(*
Nazwa:			FB_State
Opis:			Generowanie stanów 
Wersja:			v1.0
Data:			2020-04-14
Autor:			DP
Urzadzenia:		
Konfiguracja:	
Info: 
*)

FUNCTION_BLOCK FB_State
VAR_INPUT
	eState							:E_Station;						//Stan ogólny bloku
	bRun							:BOOL;							//Rozkad cyklu	
	eGripperScrewerRunningState		:E_GripperScrewer; 				//Stan zakręcarki szczekowej							
	//eRollerScrewerRunningState		:E_RollerScrewer; 				//Stan zakręcarki rolkowej						
	eCheckerRunningState			:E_CheckerState; 				//Stan sprawdzania
	eEntranceGatesRunningState		:E_EntranceGatesState;			//Stan szlabanów
	eCatchRunningState				:E_CatchStationState;			//Stan wewnętrzny
	eCapPushingRunningState			:E_CapPushingState;				//Stan wbijaka
	eMassHeatingRunningState		:E_MassHeatingState;			//Stan grzania
	eConveyorRunningState			:E_ConveyorState;				//Stan transprterów
	eFormsDragingRunningState 		:E_DragStationState;				//Stan przeciągania zwykłego
	eFormsDragingPneumRunningState	:E_DragStationStatePneum;
	eLidSealingRunningState			:E_LidSealing;					//Stan zgrzewania
	eLidFeederRunningState			:E_LidFeederState;				//Stan platynkowania
	//eWheelRunningState				:E_WheelState;					//Stan kola
	eDispencerRunningState			:E_DispencerState;				//Stan dozowników
	eDispencerLifterRunningState	:E_DispencerLifterState;		//Stan podnośnikow
	eCapFeederRobotRunningState		:E_RobotMovState;				//Stan robota
	eWeightRunningState				:E_WeightState;	
	eWeightLiftRunningState			:E_WeightLiftStationState	;	//Stan wagi		
	eBottleSorterRunningState		:E_BottleFeederState;			// Stan podajnik opakowań		 
	eCapFeederRunningState			:E_CapFeederState;				//Stan podajnika nasadek			
	eWickFeederRunningState			:E_WickFeederState;
END_VAR
VAR_OUTPUT
	sStateDesc						:STRING;
	iState							:INT;							//Stan ogólny bloku
END_VAR
VAR
	iC: INT;
	i: E_DispencerState;
	ic2: INT;
	ic3: INT;
	ic4: INT;
END_VAR


IF 	eState = 0 THEN // eDisabled := 0,	
	sStateDesc := 'Wyłączona';
ELSIF 	eState = 1 THEN // eAborted := 1,
	sStateDesc := 'Bezpieczne zatrzymanie';
ELSIF 	eState = 2 THEN // eAborting := 2,  
	sStateDesc := 'Bezpieczne zatrzymywanie';
ELSIF 	eState = 3 THEN // eError := 3,	
	sStateDesc := 'Błąd';
ELSIF 	eState = 4 THEN // eResetting := 4,	
	sStateDesc := 'Resetowanie';
ELSIF 	eState = 5 THEN // eManualMovement := 5, 
	sStateDesc := 'Tryb serwisowy';
ELSIF 	eState = 6 THEN // eHoming := 6,
	sStateDesc := 'Bazowanie';
ELSIF 	eState = 7 THEN // eHomingDone := 7,
	sStateDesc := 'Koniec bazowania';	
ELSIF 	eState = 8 THEN // ePreparingToReady := 8,	
	sStateDesc := 'Przygotowanie do gotowości';
ELSIF 	eState = 9 THEN // ePreparingToDisable := 9,
	sStateDesc := 'Przygotowanie do wyłączenia';	
ELSIF 	eState = 10 THEN // eReady	:= 10,
	sStateDesc := 'Gotowa';	
ELSIF 	eState = 11 THEN // eStopping := 11,
	sStateDesc := 'Zatrzymywanie';	
ELSIF 	eState = 12 THEN // eStarting := 12,
	sStateDesc := 'Uruchamianie';  
ELSIF 	eState = 13 THEN // eRunning := 13		
	sStateDesc := 'Praca';
END_IF

IF eState = 13 OR bRun THEN
	GripperScrewer();
	BottleSorter();
	RollerScrewer();	
	EntranceGates();
	CatchStation();
	MassHeating();
	Conveyor();
	CapFeeder();
	Checker();
	Dispencer();
	DispencerLifter();
	Robot();
	Weight();
	WeightLift();
	Drag();
	DragPneum();
	LidFeeder();
	LidSealing();
	WickFeeder();
END_IF

iState := eState;

ACTION BottleSorter:

IF eBottleSorterRunningState  = 1 THEN 
	sStateDesc := 'Błąd';	
ELSIF eBottleSorterRunningState  = 2 THEN 
	sStateDesc := 'Gotowa';	
ELSIF eBottleSorterRunningState  = 3 THEN 
	sStateDesc := 'Bazowanie';	
ELSIF eBottleSorterRunningState  = 4 THEN 
	sStateDesc := 'Koniec bazowania';	
ELSIF eBottleSorterRunningState  = 5 THEN 
	sStateDesc := 'Tryb ręczny';
ELSIF eBottleSorterRunningState  = 60 THEN 
	sStateDesc := 'Przygotowanie do ruchu';	
ELSIF eBottleSorterRunningState  = 70 THEN 
	sStateDesc := 'Zamknięcie bramki lewej';	
ELSIF eBottleSorterRunningState  = 80 THEN 
	sStateDesc := 'Przejazd do pobrania';	
ELSIF eBottleSorterRunningState  = 90 THEN 
	sStateDesc := 'Zamykanie chwytaka';	
ELSIF eBottleSorterRunningState  = 100 THEN 
	sStateDesc := 'Otwarcie bramki prawej';	
ELSIF eBottleSorterRunningState  = 110 THEN 
	sStateDesc := 'Przejazd nad formatke';	
ELSIF eBottleSorterRunningState  = 120 THEN 
	sStateDesc := 'Zamknięcie bramki lewej';	
ELSIF eBottleSorterRunningState  = 130 THEN 
	sStateDesc := 'Zamknięcie docisku';	
ELSIF eBottleSorterRunningState  = 140 THEN 
	sStateDesc := 'Wkładanie opakowania';	
ELSIF eBottleSorterRunningState  = 150 THEN 
	sStateDesc := 'Otwieranie chwytaka';
ELSIF eBottleSorterRunningState  = 160 THEN 
	sStateDesc := 'Powrót do pozycji gotowości';
ELSIF eBottleSorterRunningState  = 170 THEN 
	sStateDesc := 'Wypuszczanie formatki';
		
END_IF
END_ACTION

ACTION CapFeeder:
IF eCapFeederRunningState = 1 THEN
	sStateDesc := 'Gotowy';
ELSIF eCapFeederRunningState = 2 THEN
	sStateDesc := 'Niski poziom zamknięć';
ELSIF eCapFeederRunningState = 3 THEN
	sStateDesc := 'Praca';
ELSIF eCapFeederRunningState = 4 THEN
	sStateDesc := 'Zapełniony';
END_IF
END_ACTION

ACTION CapPushing:
IF eCapPushingRunningState = 1 THEN
	sStateDesc := 'Gotowy';
ELSIF eCapPushingRunningState = 2 THEN
	sStateDesc := 'Wbijanie';
ELSIF eCapPushingRunningState = 3 THEN
	sStateDesc := 'Przyciskanie';	
ELSIF eCapPushingRunningState = 4 THEN
	sStateDesc := 'Wbito';		
ELSIF eCapPushingRunningState = 5 THEN
	sStateDesc := 'Podnoszenie';									
END_IF
END_ACTION

ACTION CatchStation:
IF eCatchRunningState = 1 THEN
	sStateDesc := 'Błąd';
ELSIF eCatchRunningState = 2 THEN
	sStateDesc := 'Tryb serwisowy';
ELSIF eCatchRunningState = 4 THEN
	sStateDesc := 'Bazowanie';	
ELSIF eCatchRunningState = 5 THEN
	sStateDesc := 'Koniec bazownia';		
ELSIF eCatchRunningState = 6 THEN
	sStateDesc := 'Gotowość';			
ELSIF eCatchRunningState = 7 THEN
	sStateDesc := 'Chwytanie';				
ELSIF eCatchRunningState = 8 THEN
	sStateDesc := 'Chwycono';					
ELSIF eCatchRunningState = 9 THEN
	sStateDesc := 'Przygotowanie do wyłączenia';	
ELSIF eCatchRunningState = 10 THEN
	sStateDesc := 'Nie chwycono';					
END_IF
END_ACTION

ACTION Checker:
IF eCheckerRunningState = 1 THEN
	sStateDesc := 'Blad';
ELSIF eCheckerRunningState = 2 THEN
	sStateDesc := 'Tryb serwisowy';	
ELSIF eCheckerRunningState = 3 THEN
	sStateDesc := 'Bazowanie';		
ELSIF eCheckerRunningState = 4 THEN
	sStateDesc := 'Koniec bazowania';			
ELSIF eCheckerRunningState = 5 THEN
	sStateDesc := 'Gotowa';				
ELSIF eCheckerRunningState = 6 THEN
	sStateDesc := 'Formatka';		
ELSIF eCheckerRunningState = 7 THEN
	sStateDesc := 'Butelka';	
ELSIF eCheckerRunningState = 8 THEN
	sStateDesc := 'Platynka OK';	
ELSIF eCheckerRunningState = 9 THEN
	sStateDesc := 'Nasadka OK';	
ELSIF eCheckerRunningState = 10 THEN
	sStateDesc := 'Nasadka NOK.';		
ELSIF eCheckerRunningState = 11 THEN
	sStateDesc := 'Przyg. do wył.';		
					
END_IF
END_ACTION

ACTION Conveyor:
(*IF eConveyorRunningState = 0 THEN //Wyłączona
	sStateDesc := 'Wyłączona';
ELSIF eConveyorRunningState = 1 THEN //Błąd
	sStateDesc := 'Bład';
ELSIF eConveyorRunningState = 2 THEN //Tryb serwisowy
	sStateDesc := 'Tryb serwisowy';	
ELSIF eConveyorRunningState = 3 THEN //Bazowanie
	sStateDesc := 'Bazowanie';		
ELSIF eConveyorRunningState = 4 THEN //Koniec bazowania
	sStateDesc := 'Koniec bazowanie';	
ELSIF eConveyorRunningState = 5 THEN //gotowość
	sStateDesc := 'Gotowa';	
ELSIF eConveyorRunningState = 6 THEN //Zatrzymywanie
	sStateDesc := 'Zatrzymywanie';	
ELSIF eConveyorRunningState = 7 THEN //Startowanie
	sStateDesc := 'Startowanie';	
ELSIF eConveyorRunningState = 8 THEN //Praca
	sStateDesc := 'Praca';				
END_IF


*)
(*
IF eConveyorRunningState = 0 THEN //Wyłączona
	sStateDesc := 'Wyłączona 123';
ELSIF eConveyorRunningState = 1 THEN //Błąd
	sStateDesc := 'Bezp. zatrzymana';
ELSIF eConveyorRunningState = 2 THEN //Tryb serwisowy
	sStateDesc := 'Bezp. zatrzymywanie';	
ELSIF eConveyorRunningState = 3 THEN //Bazowanie
	sStateDesc := 'Błąd';		
ELSIF eConveyorRunningState = 4 THEN //Koniec bazowania
	sStateDesc := 'Resetowanie błędów';	
ELSIF eConveyorRunningState = 5 THEN //gotowość
	sStateDesc := 'Tryb ręczny';	
ELSIF eConveyorRunningState = 6 THEN //Zatrzymywanie
	sStateDesc := 'Bazowanie';	
ELSIF eConveyorRunningState = 7 THEN //Startowanie
	sStateDesc := 'Koniec bazowania';	
ELSIF eConveyorRunningState = 8 THEN //Praca
	sStateDesc := 'Przyg. do wył.';	
	*)
IF eConveyorRunningState = 10 THEN //Startowanie
	sStateDesc := 'Gotowośc';	
ELSIF eConveyorRunningState = 11 THEN //Praca
	sStateDesc := 'Zatrzymywanie';	
ELSIF eConveyorRunningState = 12 THEN //Praca
	sStateDesc := 'Uruchamianie';	
ELSIF eConveyorRunningState = 13 THEN //Praca
	sStateDesc := 'Praca';

	
END_IF
END_ACTION

ACTION Dispencer:
IF eDispencerRunningState = 5 THEN
	sStateDesc := 'Gotowa';	
		ic3		:= ic3+1;		
ELSIF eDispencerRunningState = 6 THEN
	sStateDesc := 'Przyg. dozy';		
ELSIF eDispencerRunningState = 7 THEN
	sStateDesc := '1 faza';	
ELSIF eDispencerRunningState = 8 THEN
	sStateDesc := '2 faza';	
ELSIF eDispencerRunningState = 9 THEN
	sStateDesc := '3 faza';	
ELSIF eDispencerRunningState = 10 THEN
	sStateDesc := 'Koniec dozy';	
ELSIF eDispencerRunningState = 11 THEN
	sStateDesc := 'Podsys';	
ELSIF eDispencerRunningState = 12 THEN
	sStateDesc := 'Koniec pods.';	
ELSIF eDispencerRunningState = 13 THEN
	sStateDesc := 'Zasysanie';				
ELSIF eDispencerRunningState = 14 THEN
	sStateDesc := 'Podnoszenie';	
ELSIF eDispencerRunningState = 15 THEN
	sStateDesc := 'Przerywanie';			
ELSIF eDispencerRunningState = 16 THEN
	sStateDesc := 'Przyg. do wył.';	
ELSIF eDispencerRunningState = 17 THEN
	sStateDesc := 'Przeciąganie';
ELSIF eDispencerRunningState = 18 THEN
	sStateDesc := 'Przyg. do mycia';
ELSIF eDispencerRunningState = 19 THEN
	sStateDesc := 'Gotowy do mycia';
ELSIF eDispencerRunningState = 20 THEN
	sStateDesc := 'Mycie';
ELSIF eDispencerRunningState = 21 THEN
	sStateDesc := 'Koniec mycia';		
END_IF

i   := eDispencerRunningState;
END_ACTION

ACTION DispencerLifter:
IF eDispencerLifterRunningState = 1 THEN
	sStateDesc := 'Blad';
ELSIF eDispencerLifterRunningState = 2 THEN
	sStateDesc := 'Tryb serwisowy';	
ELSIF eDispencerLifterRunningState = 3 THEN
	sStateDesc := 'Bazowanie';		
ELSIF eDispencerLifterRunningState = 4 THEN
	sStateDesc := 'Koniec bazowania';			
ELSIF eDispencerLifterRunningState = 5 THEN
	sStateDesc := 'Gotowa';				
ELSIF eDispencerLifterRunningState = 6 THEN
	sStateDesc := 'Przyg. dozy';		
ELSIF eDispencerLifterRunningState = 7 THEN
	sStateDesc := '1 faza';	
ELSIF eDispencerLifterRunningState = 8 THEN
	sStateDesc := '2 faza';	
ELSIF eDispencerLifterRunningState = 9 THEN
	sStateDesc := '3 faza';	
ELSIF eDispencerLifterRunningState = 10 THEN
	sStateDesc := 'Koniec dozy';	
ELSIF eDispencerLifterRunningState = 11 THEN
	sStateDesc := 'Zasysanie';	
ELSIF eDispencerLifterRunningState = 12 THEN
	sStateDesc := 'Podnoszenie';	
ELSIF eDispencerLifterRunningState = 13 THEN
	sStateDesc := 'Wylaczanie';				
ELSIF eDispencerLifterRunningState = 14 THEN
	sStateDesc := 'Przyg. do wył.';	
ELSIF eDispencerLifterRunningState = 15 THEN
	sStateDesc := 'Przeciąganie';			
ELSIF eDispencerLifterRunningState = 16 THEN
	sStateDesc := 'Podsysanie';	
ELSIF eDispencerLifterRunningState = 17 THEN
	sStateDesc := 'Koniec podsysania';		
END_IF
END_ACTION

ACTION Drag:
IF eFormsDragingRunningState = 1 THEN 
	sStateDesc := 'Bład';
ELSIF eFormsDragingRunningState  = 2 THEN 
	sStateDesc := 'Gotowość';	
ELSIF eFormsDragingRunningState  = 3 THEN 
	sStateDesc := 'Tryb serwisowy';	
ELSIF eFormsDragingRunningState  = 4 THEN 
	sStateDesc := 'Przygotowanie do ruchu';	
ELSIF eFormsDragingRunningState  = 5 THEN 
	sStateDesc := 'Bazowanie';	
ELSIF eFormsDragingRunningState  = 6 THEN 
	sStateDesc := 'Koniec bazowania';	
ELSIF eFormsDragingRunningState  = 7 THEN 
	sStateDesc := 'Podnoszenie';	
ELSIF eFormsDragingRunningState  = 8 THEN 
	sStateDesc := 'Przyg. do przec.';	
ELSIF eFormsDragingRunningState  = 9 THEN 
	sStateDesc := 'Przeciąganie';	
ELSIF eFormsDragingRunningState  = 10 THEN 
	sStateDesc := 'Koniec Przec.';	
ELSIF eFormsDragingRunningState  = 11 THEN 
	sStateDesc := 'Zakańczanie przec.';	
ELSIF eFormsDragingRunningState  = 12 THEN 
	sStateDesc := 'Koniec zakań. przec.';	
ELSIF eFormsDragingRunningState  = 13 THEN 
	sStateDesc := 'Opuszczanie';	
ELSIF eFormsDragingRunningState  = 14 THEN 
	sStateDesc := 'Przeciągniete';	
ELSIF eFormsDragingRunningState  = 15 THEN 
	sStateDesc := 'Koniec cyklu';	
			
END_IF
END_ACTION

ACTION DragPneum:
IF eFormsDragingPneumRunningState= 1 THEN 
	sStateDesc := 'Bład';
ELSIF eFormsDragingPneumRunningState  = 2 THEN 
	sStateDesc := 'Gotowość';	
ELSIF eFormsDragingPneumRunningState  = 3 THEN 
	sStateDesc := 'Tryb serwisowy';	
ELSIF eFormsDragingPneumRunningState  = 4 THEN 
	sStateDesc := 'Przygotowanie do ruchu';	
ELSIF eFormsDragingPneumRunningState  = 5 THEN 
	sStateDesc := 'Bazowanie';	
ELSIF eFormsDragingPneumRunningState  = 6 THEN 
	sStateDesc := 'Koniec bazowania';	
ELSIF eFormsDragingPneumRunningState  = 7 THEN 
	sStateDesc := 'Podnoszenie';	
ELSIF eFormsDragingPneumRunningState  = 8 THEN 
	sStateDesc := 'Przyg. do przec.';	
ELSIF eFormsDragingPneumRunningState  = 9 THEN 
	sStateDesc := 'Przeciąganie';	
ELSIF eFormsDragingPneumRunningState  = 10 THEN 
	sStateDesc := 'Koniec Przec.';	
ELSIF eFormsDragingPneumRunningState  = 11 THEN 
	sStateDesc := 'Korekta pozycji';	
ELSIF eFormsDragingPneumRunningState  = 12 THEN 
	sStateDesc := 'Koniec korekty';	
ELSIF eFormsDragingPneumRunningState  = 13 THEN 
	sStateDesc := 'Opuszczanie';	
ELSIF eFormsDragingPneumRunningState  = 14 THEN 
	sStateDesc := 'Przeciągniete';	
ELSIF eFormsDragingPneumRunningState  = 15 THEN 
	sStateDesc := 'Koniec cyklu';					
END_IF
END_ACTION

ACTION EntranceGates:
IF eEntranceGatesRunningState = 1 THEN
	sStateDesc := 'Błąd';
ELSIF eEntranceGatesRunningState = 2 THEN
	sStateDesc := 'Tryb serwisowy';
ELSIF eEntranceGatesRunningState = 4 THEN
	sStateDesc := 'Bazowanie';	
ELSIF eEntranceGatesRunningState = 5 THEN
	sStateDesc := 'Koniec bazownia';		
ELSIF eEntranceGatesRunningState = 6 THEN
	sStateDesc := 'Gotowość';			
ELSIF eEntranceGatesRunningState = 8 THEN
	sStateDesc := 'Wjazd 2 ';				
ELSIF eEntranceGatesRunningState = 9 THEN
	sStateDesc := 'Wjazd 1';					
ELSIF eEntranceGatesRunningState = 11 THEN
	sStateDesc := 'Czekanie';						
ELSIF eEntranceGatesRunningState = 12 THEN
	sStateDesc := 'Wyjazd 2';							
ELSIF eEntranceGatesRunningState = 13 THEN
	sStateDesc := 'Wyjazd 1';	
ELSIF eEntranceGatesRunningState = 14 THEN
	sStateDesc := 'Blokowanie';	
ELSIF eEntranceGatesRunningState = 15 THEN
	sStateDesc := 'Otwieranie';	
ELSIF eEntranceGatesRunningState = 16 THEN
	sStateDesc := 'Otwarty';	
ELSIF eEntranceGatesRunningState = 17 THEN
	sStateDesc := 'Przygotowanie do gotowości';	
ELSIF eEntranceGatesRunningState = 18 THEN
	sStateDesc := 'Przygotowanie do wyłączenia';	
ELSIF eEntranceGatesRunningState = 19 THEN
	sStateDesc := 'Przeciąganie do środka';	
ELSIF eEntranceGatesRunningState = 20 THEN
	sStateDesc := 'Przeciągnięto do środka';			
END_IF
END_ACTION

ACTION GripperScrewer:
IF eGripperScrewerRunningState = 1 THEN
	sStateDesc := 'Gotowa';
ELSIF eGripperScrewerRunningState = 2 THEN
	sStateDesc := 'Przejazd do wbijania';
ELSIF eGripperScrewerRunningState = 3 THEN
	sStateDesc := 'Przejazd do zakrecania';	
ELSIF eGripperScrewerRunningState = 4 THEN
	sStateDesc := 'Wcisnieto';		
ELSIF eGripperScrewerRunningState = 5 THEN
	sStateDesc := 'Szukanie gwintu';			
ELSIF eGripperScrewerRunningState = 6 THEN
	sStateDesc := 'Zakrecanie';				
ELSIF eGripperScrewerRunningState = 7 THEN
	sStateDesc := 'Podnoszenie';					
ELSIF eGripperScrewerRunningState = 8 THEN
	sStateDesc := 'Zakrecono';						
ELSIF eGripperScrewerRunningState = 9 THEN
	sStateDesc := 'Niezakręcono';							
ELSIF eGripperScrewerRunningState = 10 THEN
	sStateDesc := 'Przytrzymywanie';			
END_IF
END_ACTION

ACTION LidFeeder:
IF eLidFeederRunningState = 1 THEN
	sStateDesc := 'Blad';
ELSIF eLidFeederRunningState = 2 THEN
	sStateDesc := 'Tryb serwisowy';	
ELSIF eLidFeederRunningState = 3 THEN
	sStateDesc := 'Bazowanie';		
ELSIF eLidFeederRunningState = 4 THEN
	sStateDesc := 'Koniec bazowania';			
ELSIF eLidFeederRunningState = 5 THEN
	sStateDesc := 'Nagrzewanie';				
ELSIF eLidFeederRunningState = 6 THEN
	sStateDesc := 'Gotowa';		
ELSIF eLidFeederRunningState = 7 THEN
	sStateDesc := 'Zasysanie';	
ELSIF eLidFeederRunningState = 8 THEN
	sStateDesc := 'Nakładanie';	
ELSIF eLidFeederRunningState = 9 THEN
	sStateDesc := 'Nakładanie 2';	
ELSIF eLidFeederRunningState = 10 THEN
	sStateDesc := 'Zgrzewanie';	
ELSIF eLidFeederRunningState = 11 THEN
	sStateDesc := 'Odlożona';	
ELSIF eLidFeederRunningState = 12 THEN
	sStateDesc := 'Podnoszenie';	
ELSIF eLidFeederRunningState = 13 THEN
	sStateDesc := 'Przyg.do wyłączenia';						
END_IF
END_ACTION

ACTION LidSealing:

IF eLidSealingRunningState = 1 THEN
	sStateDesc := 'Nagrzewanie';
ELSIF eLidSealingRunningState = 2 THEN
	sStateDesc := 'Gotowa';	
ELSIF eLidSealingRunningState = 3 THEN
	sStateDesc := 'Zgrzewanie';		
ELSIF eLidSealingRunningState = 4 THEN
	sStateDesc := 'Grzanie';			
ELSIF eLidSealingRunningState = 5 THEN
	sStateDesc := 'Zgrzano';				
ELSIF eLidSealingRunningState = 6 THEN
	sStateDesc := 'Podnoszenie';							
END_IF
END_ACTION

ACTION MassHeating:
IF eMassHeatingRunningState = 1 THEN //Grzanie
	sStateDesc := 'Grzanie';
ELSIF eMassHeatingRunningState = 2 THEN //Gotowość
	sStateDesc := 'Utrzymywanie temp.';	
ELSIF eMassHeatingRunningState = 3 THEN //Chłodzenie
	sStateDesc := 'Chłodzenie';					
END_IF
END_ACTION

ACTION Robot:
IF eCapFeederRobotRunningState = 1 THEN
	sStateDesc := 'Pobieranie';
ELSIF eCapFeederRobotRunningState = 2 THEN
	sStateDesc := 'Pobrano';
ELSIF eCapFeederRobotRunningState = 3 THEN
	sStateDesc := 'Odkładanie';	
ELSIF eCapFeederRobotRunningState = 4 THEN
	sStateDesc := 'Pobrano';		
ELSIF eCapFeederRobotRunningState = 5 THEN
	sStateDesc := 'Odrzucanie';			
ELSIF eCapFeederRobotRunningState = 6 THEN
	sStateDesc := 'Odrzucono';				
ELSIF eCapFeederRobotRunningState = 7 THEN
	sStateDesc := 'Do start Inkjet';	
ELSIF eCapFeederRobotRunningState = 8 THEN
	sStateDesc := 'Start Inkjet';		
ELSIF eCapFeederRobotRunningState = 9 THEN
	sStateDesc := 'Do stop Inkjet';		
ELSIF eCapFeederRobotRunningState = 10 THEN
	sStateDesc := 'Stop Inkjet';		
ELSIF eCapFeederRobotRunningState = 11 THEN
	sStateDesc := 'Przerywanie';		
ELSIF eCapFeederRobotRunningState = 12 THEN
	sStateDesc := 'Powrót do gotowości';		
ELSIF eCapFeederRobotRunningState = 13 THEN
	sStateDesc := 'Pobieranie po Estopie';						
END_IF
END_ACTION

ACTION RollerScrewer:
(*IF eRollerScrewerRunningState = 1 THEN
	sStateDesc := 'Gotowa';
ELSIF eRollerScrewerRunningState = 2 THEN
	sStateDesc := 'Wciskanie';
ELSIF eRollerScrewerRunningState = 3 THEN
	sStateDesc := '';	
ELSIF eRollerScrewerRunningState = 4 THEN
	sStateDesc := 'Wcisnieto';		
ELSIF eRollerScrewerRunningState = 5 THEN
	sStateDesc := 'Szukanie gwintu';			
ELSIF eRollerScrewerRunningState = 6 THEN
	sStateDesc := 'Zakrecanie';				
ELSIF eRollerScrewerRunningState = 7 THEN
	sStateDesc := 'Podnoszenie';					
ELSIF eRollerScrewerRunningState = 8 THEN
	sStateDesc := 'Zakrecono';						
ELSIF eRollerScrewerRunningState = 9 THEN
	sStateDesc := 'Niezakręcono';							
ELSIF eRollerScrewerRunningState = 10 THEN
	sStateDesc := 'Przytrzymywanie';			
END_IF

*)
END_ACTION

ACTION Weight:
IF  eWeightRunningState = 1 THEN
	sStateDesc := 'Gotowa';	
ELSIF eWeightRunningState = 2 THEN
	sStateDesc := 'Ważenie';		
ELSIF eWeightRunningState = 3 THEN
	sStateDesc := 'Koniec ważenia';					
END_IF
END_ACTION

ACTION WeightLift:
IF  eWeightLiftRunningState	 = 10 THEN
	sStateDesc := 'Gotowa';	
ELSIF eWeightLiftRunningState	= 20 THEN
	sStateDesc := 'Przyg do magazynowania formatek';		
ELSIF eWeightLiftRunningState	 = 30 THEN
	sStateDesc := 'Czekanie na formatki';		
ELSIF eWeightLiftRunningState	 = 40 THEN
	sStateDesc := 'Rozpoczęcie ważenia';		
ELSIF eWeightLiftRunningState	 = 50 THEN
	sStateDesc := 'Ważenie';		
ELSIF eWeightLiftRunningState	 = 60 THEN
	sStateDesc := 'Opuszczanie wideł';		
ELSIF eWeightLiftRunningState	 = 70 THEN
	sStateDesc := 'Wypuszczanie formatek';		
ELSIF eWeightLiftRunningState	 = 80 THEN
	sStateDesc := 'Cykl skończony';			
END_IF
END_ACTION

ACTION Wheel:
(*IF eWheelRunningState = 1 THEN
	sStateDesc := 'Blad';
ELSIF eWheelRunningState = 2 THEN
	sStateDesc := 'Tryb serwisowy';	
ELSIF eWheelRunningState = 3 THEN
	sStateDesc := 'Bazowanie';		
ELSIF eWheelRunningState = 4 THEN
	sStateDesc := 'Koniec bazowania';			
ELSIF eWheelRunningState = 5 THEN
	sStateDesc := 'Gotowa';				
ELSIF eWheelRunningState = 6 THEN
	sStateDesc := 'Obracanie';		
ELSIF eWheelRunningState = 7 THEN
	sStateDesc := 'Koniec obracania';	
ELSIF eWheelRunningState = 8 THEN
	sStateDesc := 'Przerywanie';	
ELSIF eWheelRunningState = 9 THEN
	sStateDesc := 'Obracanie 2';	
ELSIF eWheelRunningState = 10 THEN
	sStateDesc := 'Przygtowanie go obr.';						
END_IF
*)
END_ACTION

ACTION WickFeeder:
IF eWickFeederRunningState = 1 THEN
	sStateDesc := 'Blad';
ELSIF eWickFeederRunningState = 2 THEN
	sStateDesc := 'Tryb serwisowy';	
ELSIF eWickFeederRunningState = 3 THEN
	sStateDesc := 'Bazowanie';		
ELSIF eWickFeederRunningState = 4 THEN
	sStateDesc := 'Koniec bazowania';			
ELSIF eWickFeederRunningState = 5 THEN
	sStateDesc := 'Nagrzewanie';				
ELSIF eWickFeederRunningState = 6 THEN
	sStateDesc := 'Gotowa';		
ELSIF eWickFeederRunningState = 7 THEN
	sStateDesc := 'Zasysanie';	
ELSIF eWickFeederRunningState = 8 THEN
	sStateDesc := 'Nakładanie';	
ELSIF eWickFeederRunningState = 9 THEN
	sStateDesc := 'Nakładanie 2';	
ELSIF eWickFeederRunningState = 10 THEN
	sStateDesc := 'Zgrzewanie';	
ELSIF eWickFeederRunningState = 11 THEN
	sStateDesc := 'Odlożona';	
ELSIF eWickFeederRunningState = 12 THEN
	sStateDesc := 'Podnoszenie';	
ELSIF eWickFeederRunningState = 13 THEN
	sStateDesc := 'Przyg.do wyłączenia';						
END_IF
END_ACTION

END_FUNCTION_BLOCK

(* stored: Version 1.1.0.1, ProductVersion 3.1.4026.13, FileIdentifier ad518b7a601e026328333af0796355303fe11301, FileSignature 60e10ee35d6b33f48ca86aef51c57dd6abd1697db294bf5aa15792f1a1ae46f23914db9fdca0a0d150af17467c52b12ec4dd072130535344b35785a7bf7b407df71863cf97c01a0254d2a1ced1a90340da5190389cde1fffb90f35d5ceaee9181483c8bdb0bd3b079e49ea14cfc6e8431bbda9dd9a841e6826bcbfb79f2ebd0643b705f1cf5d113c953e35d7fa08c9a7e926fb1e825f76a5e44a5ff9c20b61350347d8e3febf6cb136392e45c5021a7b6448ab274f621a57db8adf5bd0aed333345249a2570f5e0020e09921aa4d0d1afd2e3482fe69ed546b5c92dbe5e90e7c388408e9426b9b134d8b985d62087c1f422421f9527085252ae8e8b482851bf0
   POU FB_State: Id {d25e2381-bc79-447e-b5b9-6f9909e0fb03}, SpecialFunc None
   Action BottleSorter: Id {f0ea1636-2b3a-4443-bf77-44c5ded54e1d}
   Action CapFeeder: Id {1043dc8d-2b4e-4665-8ebf-b7546e2805b1}
   Action CapPushing: Id {a1bef585-5276-45d7-bb07-d5f2b732c87b}
   Action CatchStation: Id {cb4e54a8-9f6a-415f-ac70-42f554f100d8}
   Action Checker: Id {599702df-23bc-4a54-aa16-c2c9319452d5}
   Action Conveyor: Id {5eca993b-3dc9-4c6a-bcb1-7d8ad1247098}
   Action Dispencer: Id {52a1e068-405d-483f-a564-78dbba995273}
   Action DispencerLifter: Id {76f1a88b-d87d-45c7-ab64-611e39e5de61}
   Action Drag: Id {78b127c1-d125-4c70-9208-8a06229f2393}
   Action DragPneum: Id {1effa267-9c2c-436c-8e1e-9702fe3cb432}
   Action EntranceGates: Id {c28ba12a-43ce-4552-9438-e2b61619ee10}
   Action GripperScrewer: Id {f056e7eb-8164-4ee0-a924-78e18faa6b64}
   Action LidFeeder: Id {702b5b85-0271-4a67-877e-883d390847e5}
   Action LidSealing: Id {bcb1c7e0-83a1-41f0-9def-433f7c3cefa3}
   Action MassHeating: Id {5245ca94-78eb-4417-937f-884da6d45135}
   Action Robot: Id {0b962ee6-618b-427f-b6af-b548169c223f}
   Action RollerScrewer: Id {fa2c9ea7-fd4b-40ad-9b3e-8730876e2e12}
   Action Weight: Id {c5ffa6d6-d997-4b96-89df-b53e5da23b7e}
   Action WeightLift: Id {457685c7-45cd-4f8e-b312-2609c933b50a}
   Action Wheel: Id {5a6851c8-cea7-47bf-9db1-004807d05988}
   Action WickFeeder: Id {c56f7f61-74c3-4960-93d8-a4e6db8e737a} *)
